// TIA Portal V20 export
DATA_BLOCK "Simulation"   // DB203
TITLE = Simulation
// Simulation data
// stored: MemoryReserve 100
   VAR
      simHmiRotaryAxis : Array[0..49] of "LER_typeSimRotaryAxis";
      simHmiLinearAxis : Array[0..49] of "LER_typeSimLinearAxis";
      data : "LAF_typeSimulation";
   END_VAR
BEGIN
   data.simitActive := FALSE;
   data.simulationActiveHmi := TRUE;
   data.showSimulationButtonHmi := TRUE;
END_DATA_BLOCK
